TYPE ST_St030_IO :
STRUCT
	stIn	AT%I* : ST_St030_IO_IN;
	stOut	AT%Q* : ST_St030_IO_OUT;
END_STRUCT
END_TYPE

(* stored: Version 1.1.0.1
   DUT ST_St030_IO: Id {da33f69d-a412-4a9c-9c94-3fec797a259b} *)
